(* Logix 5000 project; controller ARS14002_PLC vendor 1 type 14 code 218 rev 30.11; software revision 30.01; part 8 of 13 *)
(* tags used below, declared in another part *)
   ARS_DERIME_AUTO : BOOL;
   ARS_Manual_Backfill : BOOL;   // **future use
   ARS_RETURN_AUTO : BOOL;
   ARS_STANDBY : BOOL;
   CP_Hi_Press_Shutoff : BOOL;
   CP_PumpUp : BOOL;
   CP_PumpUp_DN_ONS_OB : BOOL;
   CP_PumpUp_PressurePermissive : BOOL;
   CP_PumpUp_Standby_Press_SP_H : DINT;
   CP_PumpUp_Standby_Press_SP_L : DINT;
   CP_Run : BOOL;
   CP_Run_Atomize : BOOL;
   CP_Run_Standby : BOOL;
   CP_Select_Auto : BOOL;
   CP_Speed_SP_Atomize : REAL;
   CP_Speed_SP_Standby : DINT;
   CP_Start_Vent_TMR_PRE : DINT;
   FVR_800C_Auto : BOOL;
   FVR_800C_EN : BOOL;
   FVR_800C_FREQ_OUT : REAL;
   FVR_800C_PRIMARY : BOOL;
   FVR_800C_RUNNING : BOOL;
   FVR_800C_ST : BOOL;
   FVR_800D_Auto : BOOL;
   FVR_800D_EN : BOOL;
   FVR_800D_FREQ_OUT : REAL;
   FVR_800D_PRIMARY : BOOL;
   FVR_800D_RUNNING : BOOL;
   FVR_800D_ST : BOOL;
   HP_Shutoff_PerPump : REAL;
   HP_Shutoff_SPH : DINT;
   HP_Shutoff_SPL : DINT;
   IGNORE_TE_802S : BOOL;   // Don't look at TE_802
   MODE_ATOMIZE : BOOL;
   P_800_COOLDOWN_ALT_TIME : REAL;
   P_800_COOLDOWN_ALT_TIME_MS : DINT;
   P_800A_Cavit : BOOL;
   P_800A_CAVIT_CHK_TMR : TIMER;
   P_800A_CAVIT_CTR : COUNTER;
   P_800A_CAVIT_CTR_MONTH : COUNTER;
   P_800A_Cavit_Shutdown : BOOL;
   P_800A_CAVIT_TEMP_SP : DINT;
   P_800A_CAVIT_VENT_START_DLA_TMR : TIMER;
   P_800A_Cavit_Vent_TMR : TIMER;
   P_800A_COOLDOWN_ALT_TON : TIMER;
   P_800A_Hi_Press_Shutoff : BOOL;
   P_800A_Init_OK : BOOL;
   P_800A_Pre_Vent_Done : BOOL;
   P_800A_Pre_Vent_Pending : BOOL;
   P_800A_Prestart : BOOL;
   P_800A_Ready : BOOL;
   P_800A_Select_Auto_Online : BOOL;
   P_800A_Start_DLA_TMR : TIMER;
   P_800A_Start_TMR : TIMER;
   P_800A_Start_Vent_TMR : TIMER;
   P_800A_Stop_Vent_Delay : BOOL;
   P_800A_Stop_Vent_TMR : TIMER;
   P_800B_Cavit : BOOL;
   P_800B_CAVIT_CHK_TMR : TIMER;
   P_800B_CAVIT_CTR : COUNTER;
   P_800B_CAVIT_CTR_MONTH : COUNTER;
   P_800B_Cavit_Shutdown : BOOL;
   P_800B_CAVIT_TEMP_SP : DINT;
   P_800B_CAVIT_VENT_START_DLA_TMR : TIMER;
   P_800B_Cavit_Vent_TMR : TIMER;
   P_800B_COOLDOWN_ALT_TON : TIMER;
   P_800B_Hi_Press_Shutoff : BOOL;
   P_800B_Init_OK : BOOL;
   P_800B_Pre_Vent_Done : BOOL;
   P_800B_Pre_Vent_Pending : BOOL;
   P_800B_Prestart : BOOL;
   P_800B_Ready : BOOL;
   P_800B_Select_Auto_Online : BOOL;
   P_800B_Start_DLA_TMR : TIMER;
   P_800B_Start_TMR : TIMER;
   P_800B_Start_Vent_TMR : TIMER;
   P_800B_Stop_Vent_Delay : BOOL;
   P_800B_Stop_Vent_TMR : TIMER;
   P_800C : CM_DO_FVR;
   P_800C_Cavit : BOOL;
   P_800C_CAVIT_CHK_TMR : TIMER;
   P_800C_CAVIT_CTR : COUNTER;
   P_800C_CAVIT_CTR_MONTH : COUNTER;
   P_800C_Cavit_Shutdown : BOOL;
   P_800C_CAVIT_TEMP_SP : DINT;
   P_800C_CAVIT_VENT_START_DLA_TMR : TIMER;
   P_800C_Cavit_Vent_TMR : TIMER;
   P_800C_COOLDOWN_ALT_TON : TIMER;
   P_800C_Fault : BOOL;
   P_800C_Hi_Press_Shutoff : BOOL;
   P_800C_Init_OK : BOOL;
   P_800C_Pre_Vent_Done : BOOL;
   P_800C_Pre_Vent_Pending : BOOL;
   P_800C_Prestart : BOOL;
   P_800C_Ready : BOOL;
   P_800C_Start_DLA_TMR : TIMER;
   P_800C_Start_TMR : TIMER;
   P_800C_Start_Vent_TMR : TIMER;
   P_800C_Stop_Vent_Delay : BOOL;
   P_800C_Stop_Vent_TMR : TIMER;
   P_800D : CM_DO_FVR;
   P_800D_Cavit : BOOL;
   P_800D_CAVIT_CHK_TMR : TIMER;
   P_800D_CAVIT_CTR : COUNTER;
   P_800D_CAVIT_CTR_MONTH : COUNTER;
   P_800D_Cavit_Shutdown : BOOL;
   P_800D_CAVIT_TEMP_SP : DINT;
   P_800D_CAVIT_VENT_START_DLA_TMR : TIMER;
   P_800D_Cavit_Vent_TMR : TIMER;
   P_800D_COOLDOWN_ALT_TON : TIMER;
   P_800D_Fault : BOOL;
   P_800D_Hi_Press_Shutoff : BOOL;
   P_800D_Init_OK : BOOL;
   P_800D_Pre_Vent_Done : BOOL;
   P_800D_Pre_Vent_Pending : BOOL;
   P_800D_Prestart : BOOL;
   P_800D_Ready : BOOL;
   P_800D_Start_DLA_TMR : TIMER;
   P_800D_Start_Temp_SP : DINT;
   P_800D_Start_TMR : TIMER;
   P_800D_Start_Vent_TMR : TIMER;
   P_800D_Stop_Vent_Delay : BOOL;
   P_800D_Stop_Vent_TMR : TIMER;
   PDT_751 : CM_AI_SCL_ALT;
   PIDE_800 : PID_ENHANCED;
   PIDE_800_CVOper_HZ : REAL;
   PIDE_800_CVProg_HZ : REAL;
   PIDE_800_OPER_ONS : BOOL;
   PT_802A : CM_AI_SCL;
   PT_802B : CM_AI_SCL;
   PT_802C : CM_AI_SCL;
   PT_802D : CM_AI_SCL;
   PT_806 : CM_AI_SCL;
   PT_902 : CM_AI_SCL;
   PUMP_CALC_FLOW : REAL;
   PUMP_CAVIT_PRESSURE_MARGIN : REAL;   // HOW MUCH LOWER PUMP PT CAN BE THAN PT-902
   PUMP_CAVIT_PRESSURE_SP : REAL;
   PWHMI_StartAtomizing : TIMER;
   START_ATOMIZE_DURING_PUMPUP : BOOL;
   SV_802AX : CM_DO_GENERIC;
   SV_802BX : CM_DO_GENERIC;
   SV_802CX : CM_DO_GENERIC;
   SV_802DX : CM_DO_GENERIC;
   TE_802_INIT_TEMP : REAL;
   TE_802A : CM_AI_SCL;
   TE_802B : CM_AI_SCL;
   TE_802C : CM_AI_SCL;
   TE_802D : CM_AI_SCL;
   TE_803D : CM_AI_SCL;
   TE_804_INIT_TEMP : REAL;
   TE_804A : CM_AI_SCL;
   TE_804B : CM_AI_SCL;
   TE_804C : CM_AI_SCL;
   TE_804D : CM_AI_SCL;
   TEST_COOLDOWN_ALT : BOOL;
   VFD_800A_Auto : BOOL;
   VFD_800A_EN : BOOL;
   VFD_800A_ST : BOOL;
   VFD_800B_Auto : BOOL;
   VFD_800B_EN : BOOL;
   VFD_800B_ST : BOOL;
   XV_806 : CM_DO_VLV;
   XV_806_SPH_802_CLOSED : REAL;
   XV_806_SPH_802_OPEN : REAL;
   XV_806_SPL_802_CLOSED : REAL;
   XV_806_SPL_802_OPEN : REAL;
(* MainProgram, continued *)

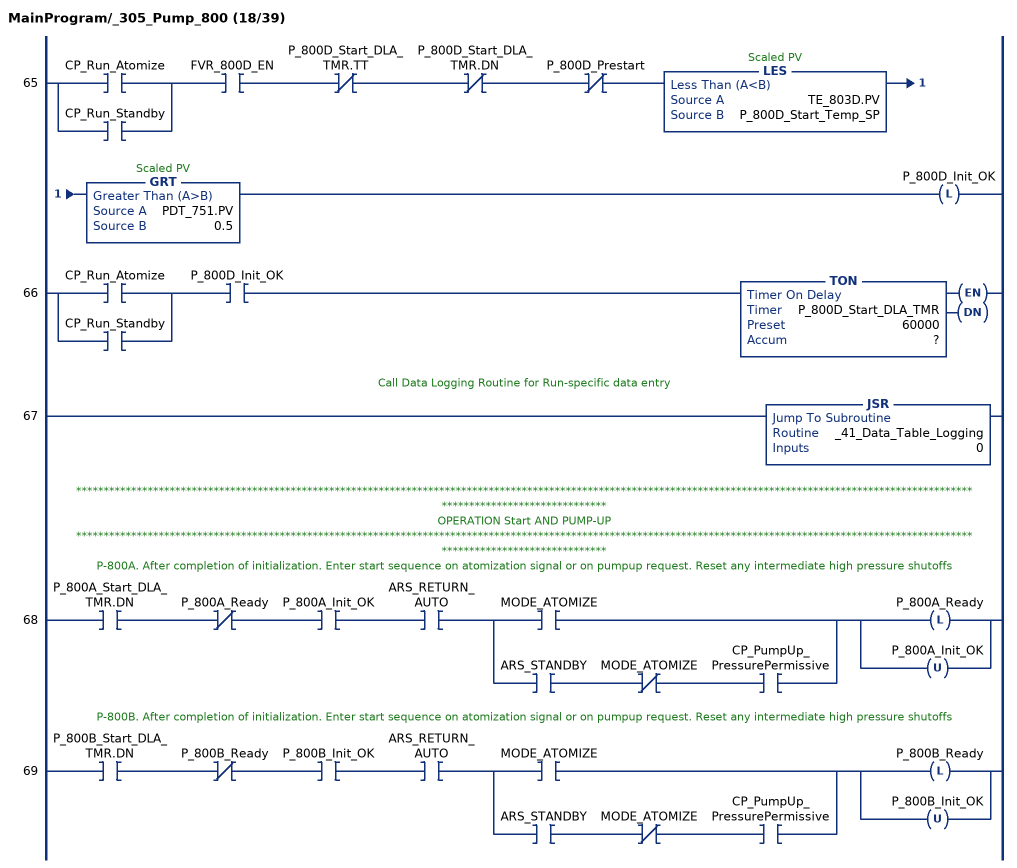
   [picture p154: MainProgram/_305_Pump_800 rungs 65-69]
   65: [XIC(CP_Run_Atomize) ,XIC(CP_Run_Standby) ]XIC(FVR_800D_EN)XIO(P_800D_Start_DLA_TMR.TT)XIO(P_800D_Start_DLA_TMR.DN)XIO(P_800D_Prestart)LES(TE_803D.PV,P_800D_Start_Temp_SP)GRT(PDT_751.PV,0.5)OTL(P_800D_Init_OK);
   66: [XIC(CP_Run_Atomize) ,XIC(CP_Run_Standby) ]XIC(P_800D_Init_OK)TON(P_800D_Start_DLA_TMR,?,?);
   // Call Data Logging Routine for Run-specific data entry
   67: JSR(_41_Data_Table_Logging,0);
   // *************************************************************************************************************************************************************************************************
   // OPERATION Start AND PUMP-UP
   // *************************************************************************************************************************************************************************************************
   // P-800A. After completion of initialization. Enter start sequence on atomization signal or on pumpup request. Reset any intermediate high pressure shutoffs
   68: XIC(P_800A_Start_DLA_TMR.DN)XIO(P_800A_Ready)XIC(P_800A_Init_OK)XIC(ARS_RETURN_AUTO)[XIC(MODE_ATOMIZE) ,XIC(ARS_STANDBY) XIO(MODE_ATOMIZE) XIC(CP_PumpUp_PressurePermissive) ][OTL(P_800A_Ready) ,OTU(P_800A_Init_OK) ];
   // P-800B. After completion of initialization. Enter start sequence on atomization signal or on pumpup request. Reset any intermediate high pressure shutoffs
   69: XIC(P_800B_Start_DLA_TMR.DN)XIO(P_800B_Ready)XIC(P_800B_Init_OK)XIC(ARS_RETURN_AUTO)[XIC(MODE_ATOMIZE) ,XIC(ARS_STANDBY) XIO(MODE_ATOMIZE) XIC(CP_PumpUp_PressurePermissive) ][OTL(P_800B_Ready) ,OTU(P_800B_Init_OK) ];
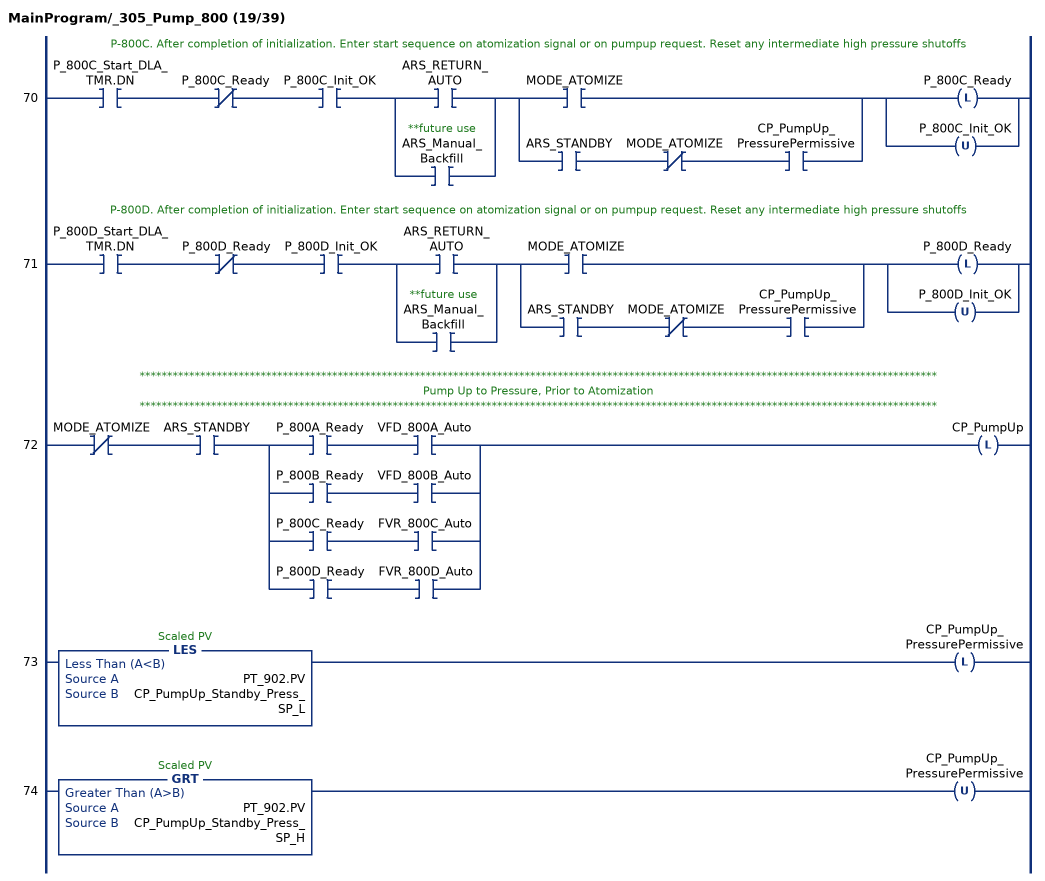
   // P-800C. After completion of initialization. Enter start sequence on atomization signal or on pumpup request. Reset any intermediate high pressure shutoffs
   70: XIC(P_800C_Start_DLA_TMR.DN)XIO(P_800C_Ready)XIC(P_800C_Init_OK)[XIC(ARS_RETURN_AUTO) ,XIC(ARS_Manual_Backfill) ][XIC(MODE_ATOMIZE) ,XIC(ARS_STANDBY) XIO(MODE_ATOMIZE) XIC(CP_PumpUp_PressurePermissive) ][OTL(P_800C_Ready) ,OTU(P_800C_Init_OK) ];
   // P-800D. After completion of initialization. Enter start sequence on atomization signal or on pumpup request. Reset any intermediate high pressure shutoffs
   71: XIC(P_800D_Start_DLA_TMR.DN)XIO(P_800D_Ready)XIC(P_800D_Init_OK)[XIC(ARS_RETURN_AUTO) ,XIC(ARS_Manual_Backfill) ][XIC(MODE_ATOMIZE) ,XIC(ARS_STANDBY) XIO(MODE_ATOMIZE) XIC(CP_PumpUp_PressurePermissive) ][OTL(P_800D_Ready) ,OTU(P_800D_Init_OK) ];
   // *************************************************************************************************************************************************
   // Pump Up to Pressure, Prior to Atomization
   // *************************************************************************************************************************************************
   72: XIO(MODE_ATOMIZE)XIC(ARS_STANDBY)[XIC(P_800A_Ready) XIC(VFD_800A_Auto) ,XIC(P_800B_Ready) XIC(VFD_800B_Auto) ,XIC(P_800C_Ready) XIC(FVR_800C_Auto) ,XIC(P_800D_Ready) XIC(FVR_800D_Auto) ]OTL(CP_PumpUp);
   73: LES(PT_902.PV,CP_PumpUp_Standby_Press_SP_L)OTL(CP_PumpUp_PressurePermissive);
   74: GRT(PT_902.PV,CP_PumpUp_Standby_Press_SP_H)OTU(CP_PumpUp_PressurePermissive);
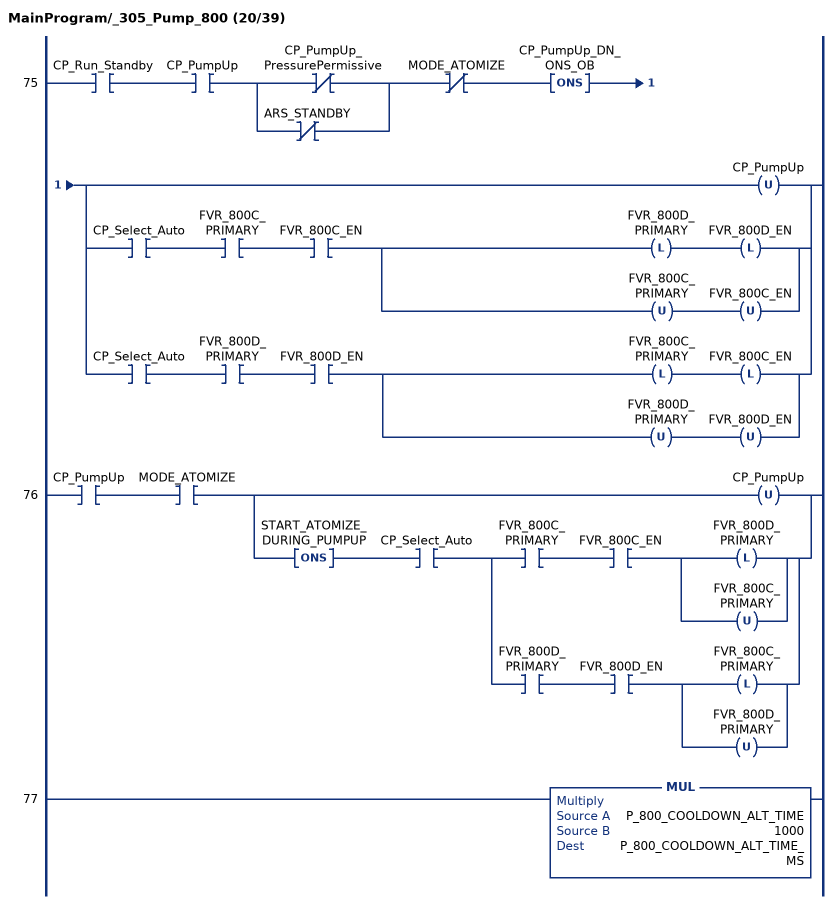
   75: XIC(CP_Run_Standby)XIC(CP_PumpUp)[XIO(CP_PumpUp_PressurePermissive) ,XIO(ARS_STANDBY) ]XIO(MODE_ATOMIZE)ONS(CP_PumpUp_DN_ONS_OB)[[OTU(CP_PumpUp) ,XIC(CP_Select_Auto) XIC(FVR_800C_PRIMARY) XIC(FVR_800C_EN) [OTL(FVR_800D_PRIMARY) OTL(FVR_800D_EN) ,OTU(FVR_800C_PRIMARY) OTU(FVR_800C_EN) ] ] ,XIC(CP_Select_Auto) XIC(FVR_800D_PRIMARY) XIC(FVR_800D_EN) [OTL(FVR_800C_PRIMARY) OTL(FVR_800C_EN) ,OTU(FVR_800D_PRIMARY) OTU(FVR_800D_EN) ] ];
   76: XIC(CP_PumpUp)XIC(MODE_ATOMIZE)[OTU(CP_PumpUp) ,ONS(START_ATOMIZE_DURING_PUMPUP) XIC(CP_Select_Auto) [XIC(FVR_800C_PRIMARY) XIC(FVR_800C_EN) [OTL(FVR_800D_PRIMARY) ,OTU(FVR_800C_PRIMARY) ] ,XIC(FVR_800D_PRIMARY) XIC(FVR_800D_EN) [OTL(FVR_800C_PRIMARY) ,OTU(FVR_800D_PRIMARY) ] ] ];
   77: MUL(P_800_COOLDOWN_ALT_TIME,1000,P_800_COOLDOWN_ALT_TIME_MS);
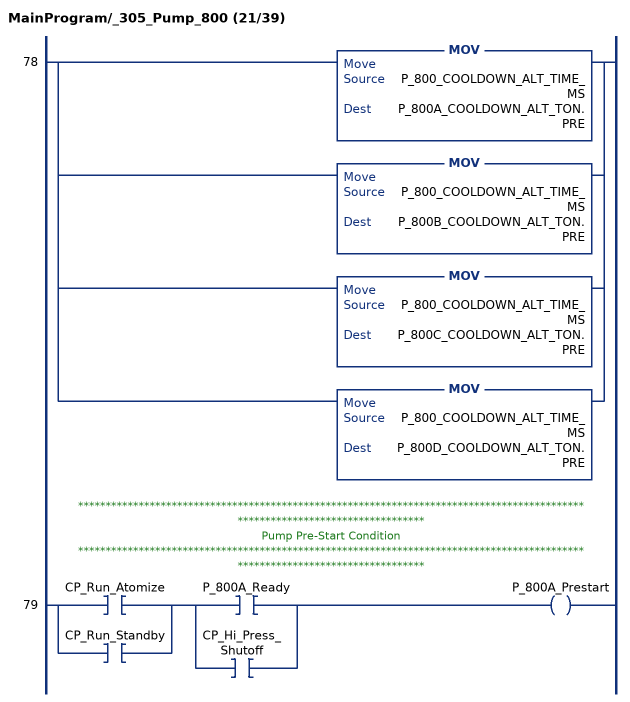
   78: [MOV(P_800_COOLDOWN_ALT_TIME_MS,P_800A_COOLDOWN_ALT_TON.PRE) ,MOV(P_800_COOLDOWN_ALT_TIME_MS,P_800B_COOLDOWN_ALT_TON.PRE) ,MOV(P_800_COOLDOWN_ALT_TIME_MS,P_800C_COOLDOWN_ALT_TON.PRE) ,MOV(P_800_COOLDOWN_ALT_TIME_MS,P_800D_COOLDOWN_ALT_TON.PRE) ];
   // ******************************************************************************************************************************
   // Pump Pre-Start Condition
   // ******************************************************************************************************************************
   79: [XIC(CP_Run_Atomize) ,XIC(CP_Run_Standby) ][XIC(P_800A_Ready) ,XIC(CP_Hi_Press_Shutoff) ]OTE(P_800A_Prestart);
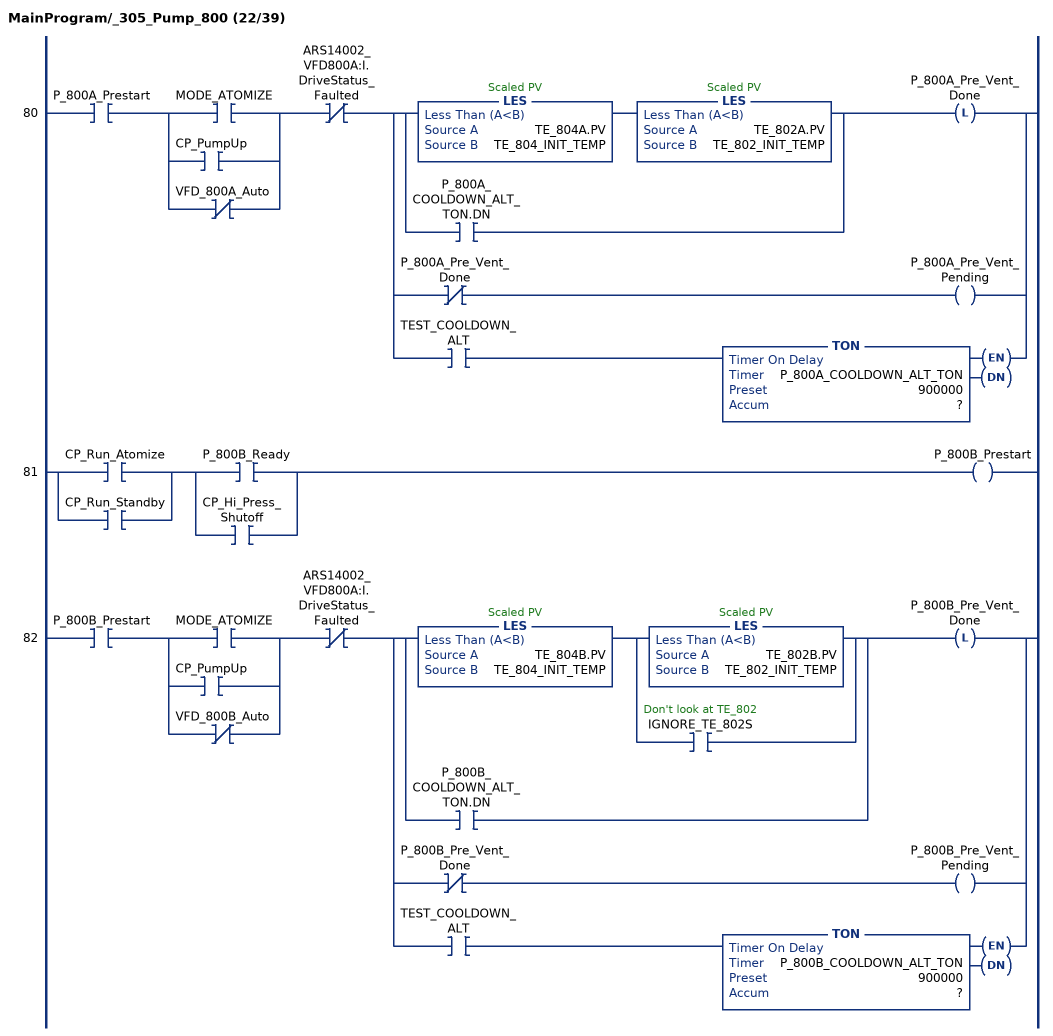
   80: XIC(P_800A_Prestart)[XIC(MODE_ATOMIZE) ,XIC(CP_PumpUp) ,XIO(VFD_800A_Auto) ]XIO(ARS14002_VFD800A:I.DriveStatus_Faulted)[[LES(TE_804A.PV,TE_804_INIT_TEMP) LES(TE_802A.PV,TE_802_INIT_TEMP) ,XIC(P_800A_COOLDOWN_ALT_TON.DN) ] OTL(P_800A_Pre_Vent_Done) ,XIO(P_800A_Pre_Vent_Done) OTE(P_800A_Pre_Vent_Pending) ,XIC(TEST_COOLDOWN_ALT) TON(P_800A_COOLDOWN_ALT_TON,?,?) ];
   81: [XIC(CP_Run_Atomize) ,XIC(CP_Run_Standby) ][XIC(P_800B_Ready) ,XIC(CP_Hi_Press_Shutoff) ]OTE(P_800B_Prestart);
   82: XIC(P_800B_Prestart)[XIC(MODE_ATOMIZE) ,XIC(CP_PumpUp) ,XIO(VFD_800B_Auto) ]XIO(ARS14002_VFD800A:I.DriveStatus_Faulted)[[LES(TE_804B.PV,TE_804_INIT_TEMP) [LES(TE_802B.PV,TE_802_INIT_TEMP) ,XIC(IGNORE_TE_802S) ] ,XIC(P_800B_COOLDOWN_ALT_TON.DN) ] OTL(P_800B_Pre_Vent_Done) ,XIO(P_800B_Pre_Vent_Done) OTE(P_800B_Pre_Vent_Pending) ,XIC(TEST_COOLDOWN_ALT) TON(P_800B_COOLDOWN_ALT_TON,?,?) ];
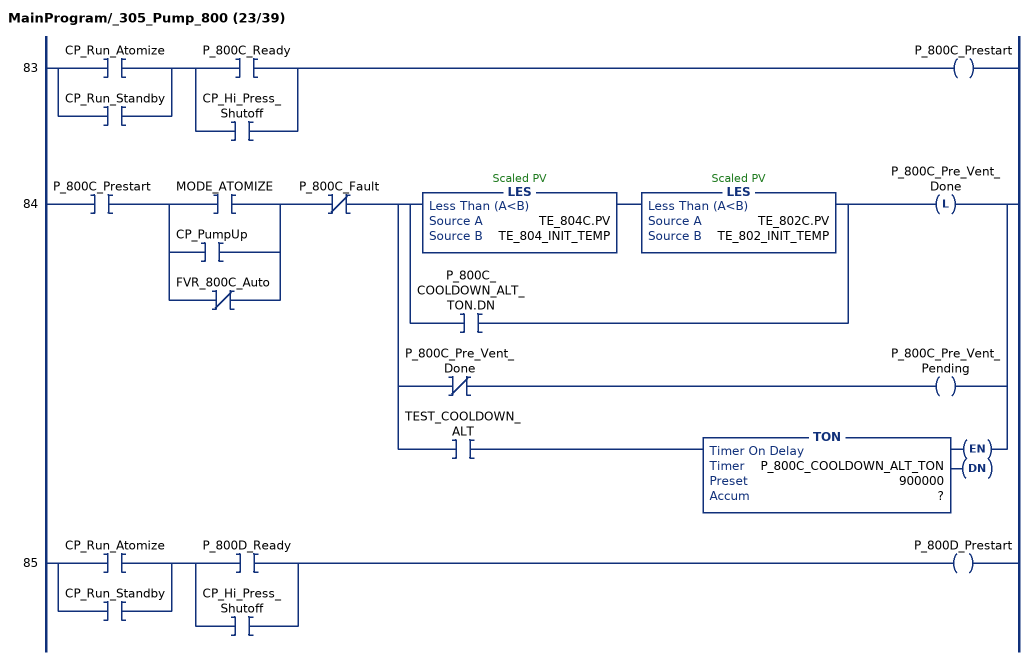
   83: [XIC(CP_Run_Atomize) ,XIC(CP_Run_Standby) ][XIC(P_800C_Ready) ,XIC(CP_Hi_Press_Shutoff) ]OTE(P_800C_Prestart);
   84: XIC(P_800C_Prestart)[XIC(MODE_ATOMIZE) ,XIC(CP_PumpUp) ,XIO(FVR_800C_Auto) ]XIO(P_800C_Fault)[[LES(TE_804C.PV,TE_804_INIT_TEMP) LES(TE_802C.PV,TE_802_INIT_TEMP) ,XIC(P_800C_COOLDOWN_ALT_TON.DN) ] OTL(P_800C_Pre_Vent_Done) ,XIO(P_800C_Pre_Vent_Done) OTE(P_800C_Pre_Vent_Pending) ,XIC(TEST_COOLDOWN_ALT) TON(P_800C_COOLDOWN_ALT_TON,?,?) ];
   85: [XIC(CP_Run_Atomize) ,XIC(CP_Run_Standby) ][XIC(P_800D_Ready) ,XIC(CP_Hi_Press_Shutoff) ]OTE(P_800D_Prestart);
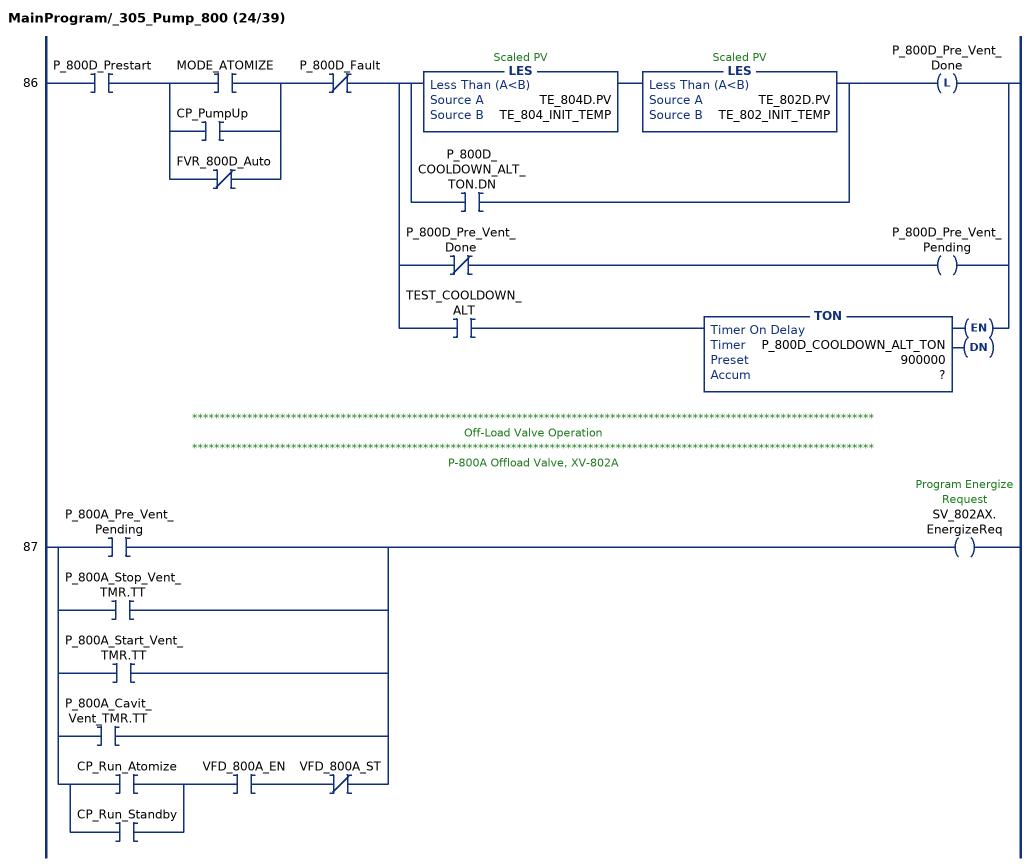
   86: XIC(P_800D_Prestart)[XIC(MODE_ATOMIZE) ,XIC(CP_PumpUp) ,XIO(FVR_800D_Auto) ]XIO(P_800D_Fault)[[LES(TE_804D.PV,TE_804_INIT_TEMP) LES(TE_802D.PV,TE_802_INIT_TEMP) ,XIC(P_800D_COOLDOWN_ALT_TON.DN) ] OTL(P_800D_Pre_Vent_Done) ,XIO(P_800D_Pre_Vent_Done) OTE(P_800D_Pre_Vent_Pending) ,XIC(TEST_COOLDOWN_ALT) TON(P_800D_COOLDOWN_ALT_TON,?,?) ];
   // ****************************************************************************************************************************
   // Off-Load Valve Operation
   // ****************************************************************************************************************************
   // P-800A Offload Valve, XV-802A
   87: [XIC(P_800A_Pre_Vent_Pending) ,XIC(P_800A_Stop_Vent_TMR.TT) ,XIC(P_800A_Start_Vent_TMR.TT) ,XIC(P_800A_Cavit_Vent_TMR.TT) ,[XIC(CP_Run_Atomize) ,XIC(CP_Run_Standby) ] XIC(VFD_800A_EN) XIO(VFD_800A_ST) ]OTE(SV_802AX.EnergizeReq);
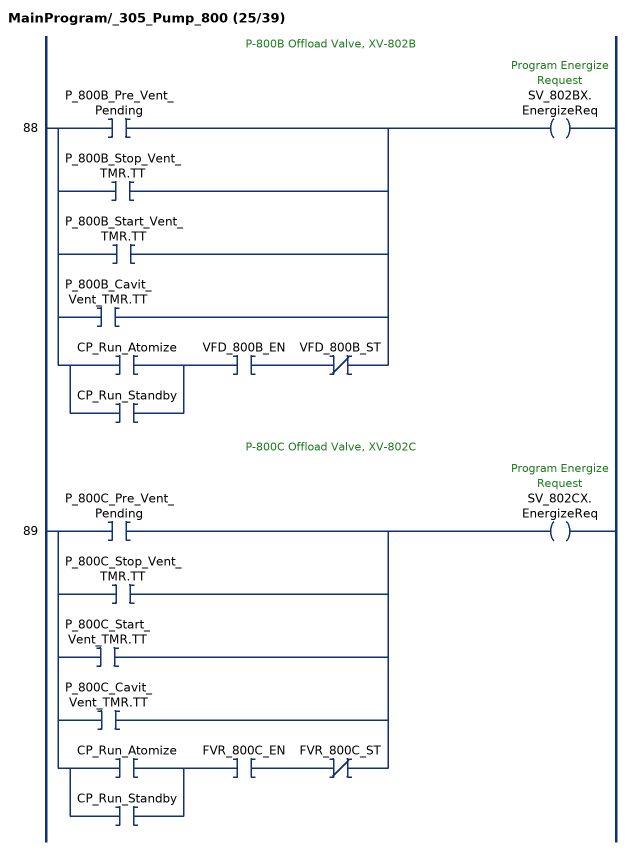
   // P-800B Offload Valve, XV-802B
   88: [XIC(P_800B_Pre_Vent_Pending) ,XIC(P_800B_Stop_Vent_TMR.TT) ,XIC(P_800B_Start_Vent_TMR.TT) ,XIC(P_800B_Cavit_Vent_TMR.TT) ,[XIC(CP_Run_Atomize) ,XIC(CP_Run_Standby) ] XIC(VFD_800B_EN) XIO(VFD_800B_ST) ]OTE(SV_802BX.EnergizeReq);
   // P-800C Offload Valve, XV-802C
   89: [XIC(P_800C_Pre_Vent_Pending) ,XIC(P_800C_Stop_Vent_TMR.TT) ,XIC(P_800C_Start_Vent_TMR.TT) ,XIC(P_800C_Cavit_Vent_TMR.TT) ,[XIC(CP_Run_Atomize) ,XIC(CP_Run_Standby) ] XIC(FVR_800C_EN) XIO(FVR_800C_ST) ]OTE(SV_802CX.EnergizeReq);
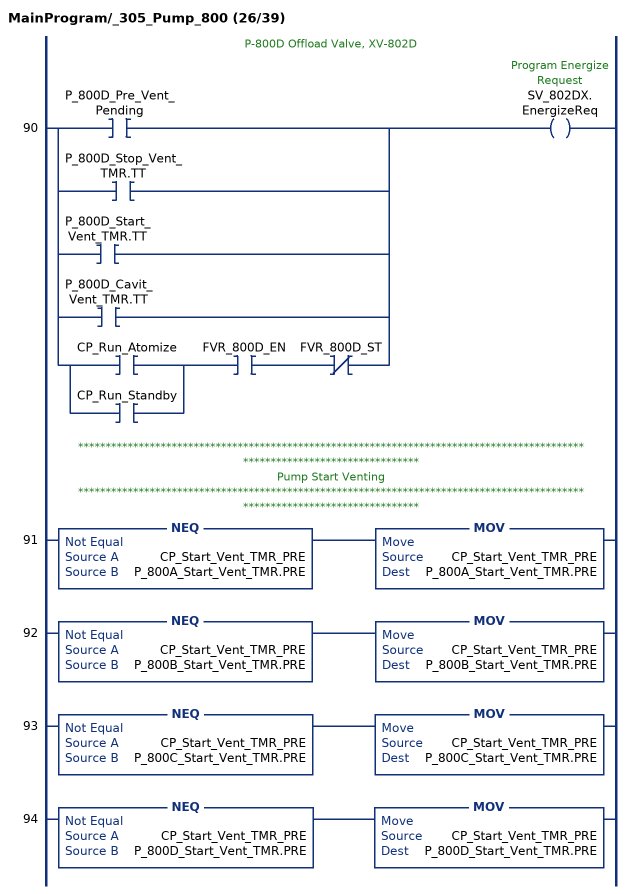
   // P-800D Offload Valve, XV-802D
   90: [XIC(P_800D_Pre_Vent_Pending) ,XIC(P_800D_Stop_Vent_TMR.TT) ,XIC(P_800D_Start_Vent_TMR.TT) ,XIC(P_800D_Cavit_Vent_TMR.TT) ,[XIC(CP_Run_Atomize) ,XIC(CP_Run_Standby) ] XIC(FVR_800D_EN) XIO(FVR_800D_ST) ]OTE(SV_802DX.EnergizeReq);
   // ****************************************************************************************************************************
   // Pump Start Venting
   // ****************************************************************************************************************************
   91: NEQ(CP_Start_Vent_TMR_PRE,P_800A_Start_Vent_TMR.PRE)MOV(CP_Start_Vent_TMR_PRE,P_800A_Start_Vent_TMR.PRE);
   92: NEQ(CP_Start_Vent_TMR_PRE,P_800B_Start_Vent_TMR.PRE)MOV(CP_Start_Vent_TMR_PRE,P_800B_Start_Vent_TMR.PRE);
   93: NEQ(CP_Start_Vent_TMR_PRE,P_800C_Start_Vent_TMR.PRE)MOV(CP_Start_Vent_TMR_PRE,P_800C_Start_Vent_TMR.PRE);
   94: NEQ(CP_Start_Vent_TMR_PRE,P_800D_Start_Vent_TMR.PRE)MOV(CP_Start_Vent_TMR_PRE,P_800D_Start_Vent_TMR.PRE);
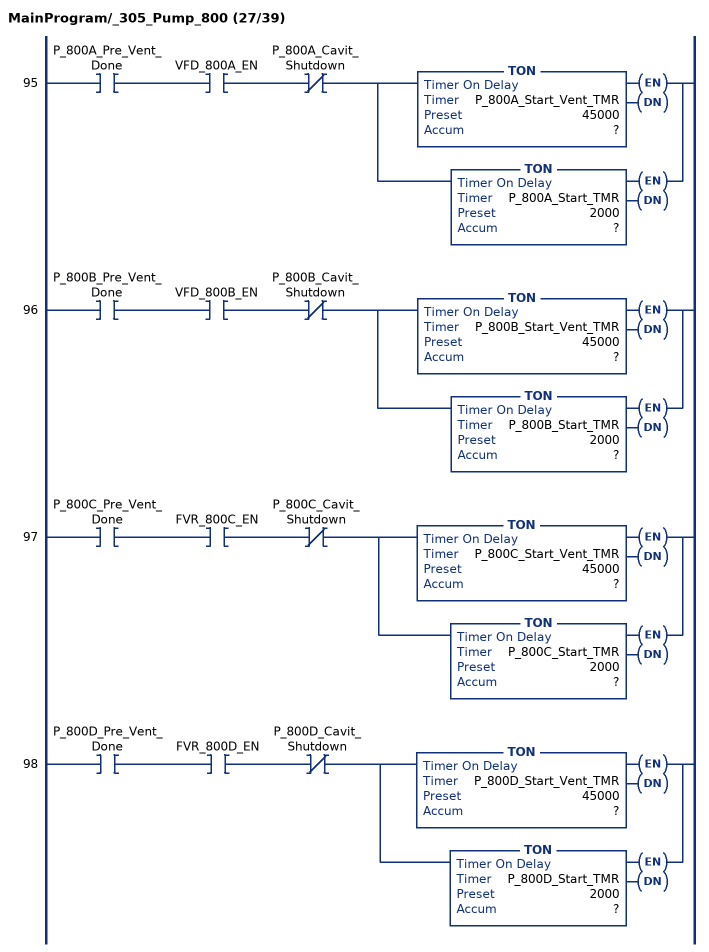
   95: XIC(P_800A_Pre_Vent_Done)XIC(VFD_800A_EN)XIO(P_800A_Cavit_Shutdown)[TON(P_800A_Start_Vent_TMR,?,?) ,TON(P_800A_Start_TMR,?,?) ];
   96: XIC(P_800B_Pre_Vent_Done)XIC(VFD_800B_EN)XIO(P_800B_Cavit_Shutdown)[TON(P_800B_Start_Vent_TMR,?,?) ,TON(P_800B_Start_TMR,?,?) ];
   97: XIC(P_800C_Pre_Vent_Done)XIC(FVR_800C_EN)XIO(P_800C_Cavit_Shutdown)[TON(P_800C_Start_Vent_TMR,?,?) ,TON(P_800C_Start_TMR,?,?) ];
   98: XIC(P_800D_Pre_Vent_Done)XIC(FVR_800D_EN)XIO(P_800D_Cavit_Shutdown)[TON(P_800D_Start_Vent_TMR,?,?) ,TON(P_800D_Start_TMR,?,?) ];
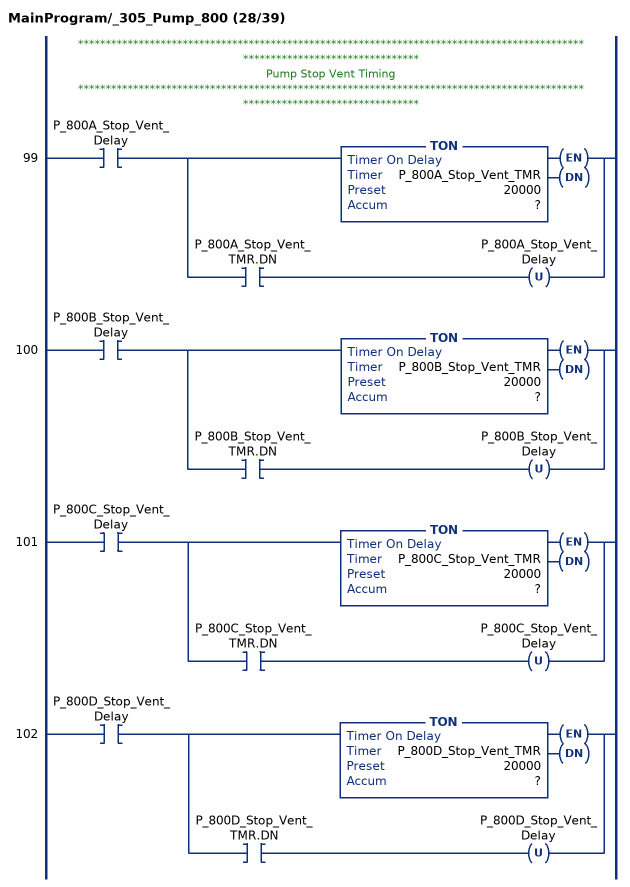
   // ****************************************************************************************************************************
   // Pump Stop Vent Timing
   // ****************************************************************************************************************************
   99: XIC(P_800A_Stop_Vent_Delay)[TON(P_800A_Stop_Vent_TMR,?,?) ,XIC(P_800A_Stop_Vent_TMR.DN) OTU(P_800A_Stop_Vent_Delay) ];
   100: XIC(P_800B_Stop_Vent_Delay)[TON(P_800B_Stop_Vent_TMR,?,?) ,XIC(P_800B_Stop_Vent_TMR.DN) OTU(P_800B_Stop_Vent_Delay) ];
   101: XIC(P_800C_Stop_Vent_Delay)[TON(P_800C_Stop_Vent_TMR,?,?) ,XIC(P_800C_Stop_Vent_TMR.DN) OTU(P_800C_Stop_Vent_Delay) ];
   102: XIC(P_800D_Stop_Vent_Delay)[TON(P_800D_Stop_Vent_TMR,?,?) ,XIC(P_800D_Stop_Vent_TMR.DN) OTU(P_800D_Stop_Vent_Delay) ];
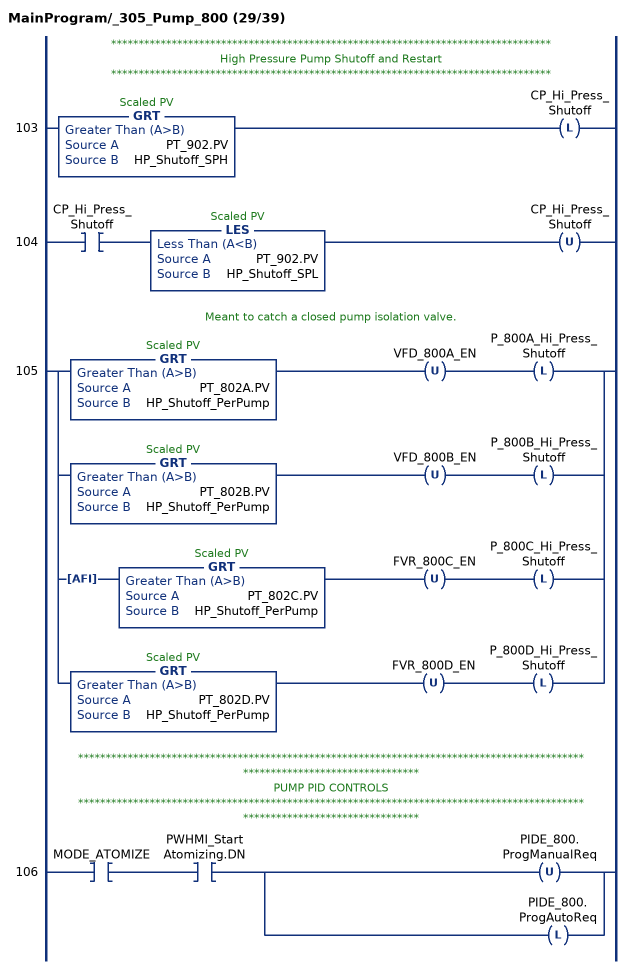
   // ********************************************************************************
   // High Pressure Pump Shutoff and Restart
   // ********************************************************************************
   103: GRT(PT_902.PV,HP_Shutoff_SPH)OTL(CP_Hi_Press_Shutoff);
   104: XIC(CP_Hi_Press_Shutoff)LES(PT_902.PV,HP_Shutoff_SPL)OTU(CP_Hi_Press_Shutoff);
   // Meant to catch a closed pump isolation valve.
   105: [GRT(PT_802A.PV,HP_Shutoff_PerPump) OTU(VFD_800A_EN) OTL(P_800A_Hi_Press_Shutoff) ,GRT(PT_802B.PV,HP_Shutoff_PerPump) OTU(VFD_800B_EN) OTL(P_800B_Hi_Press_Shutoff) ,AFI() GRT(PT_802C.PV,HP_Shutoff_PerPump) OTU(FVR_800C_EN) OTL(P_800C_Hi_Press_Shutoff) ,GRT(PT_802D.PV,HP_Shutoff_PerPump) OTU(FVR_800D_EN) OTL(P_800D_Hi_Press_Shutoff) ];
   // ****************************************************************************************************************************
   // PUMP PID CONTROLS
   // ****************************************************************************************************************************
   106: XIC(MODE_ATOMIZE)XIC(PWHMI_StartAtomizing.DN)[OTU(PIDE_800.ProgManualReq) ,OTL(PIDE_800.ProgAutoReq) ];
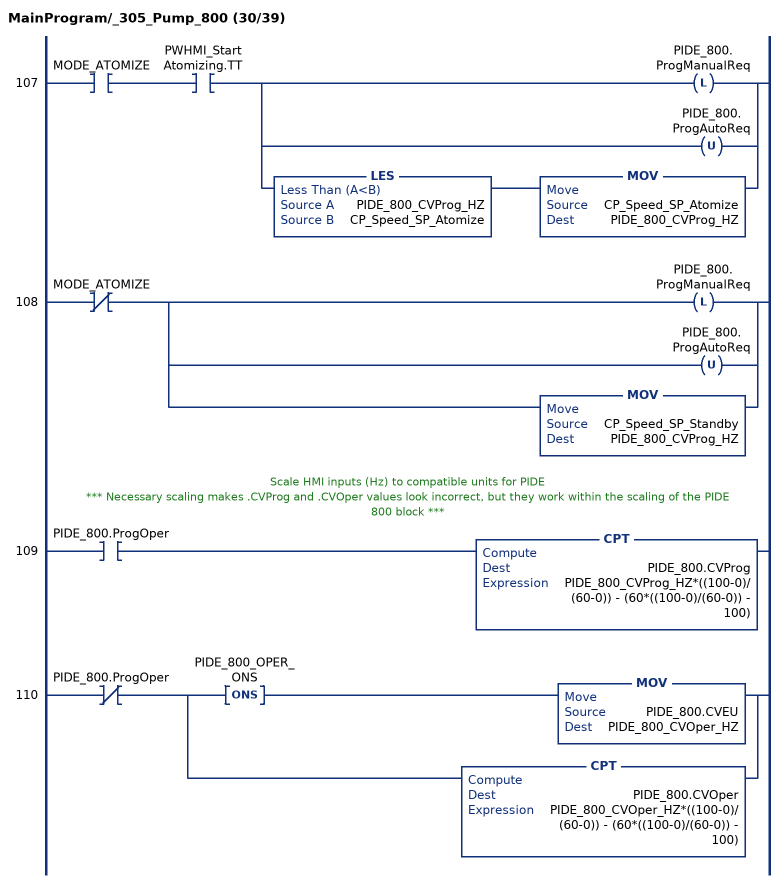
   107: XIC(MODE_ATOMIZE)XIC(PWHMI_StartAtomizing.TT)[OTL(PIDE_800.ProgManualReq) ,OTU(PIDE_800.ProgAutoReq) ,LES(PIDE_800_CVProg_HZ,CP_Speed_SP_Atomize) MOV(CP_Speed_SP_Atomize,PIDE_800_CVProg_HZ) ];
   108: XIO(MODE_ATOMIZE)[[OTL(PIDE_800.ProgManualReq) ,OTU(PIDE_800.ProgAutoReq) ] ,MOV(CP_Speed_SP_Standby,PIDE_800_CVProg_HZ) ];
   // Scale HMI inputs (Hz) to compatible units for PIDE
   // *** Necessary scaling makes .CVProg and .CVOper values look incorrect, but they work within the scaling of the PIDE 800 block ***
   109: XIC(PIDE_800.ProgOper)CPT(PIDE_800.CVProg,PIDE_800_CVProg_HZ*((100-0)/(60-0)) - (60*((100-0)/(60-0)) - 100));
   110: XIO(PIDE_800.ProgOper)[ONS(PIDE_800_OPER_ONS) MOV(PIDE_800.CVEU,PIDE_800_CVOper_HZ) ,CPT(PIDE_800.CVOper,PIDE_800_CVOper_HZ*((100-0)/(60-0)) - (60*((100-0)/(60-0)) - 100)) ];
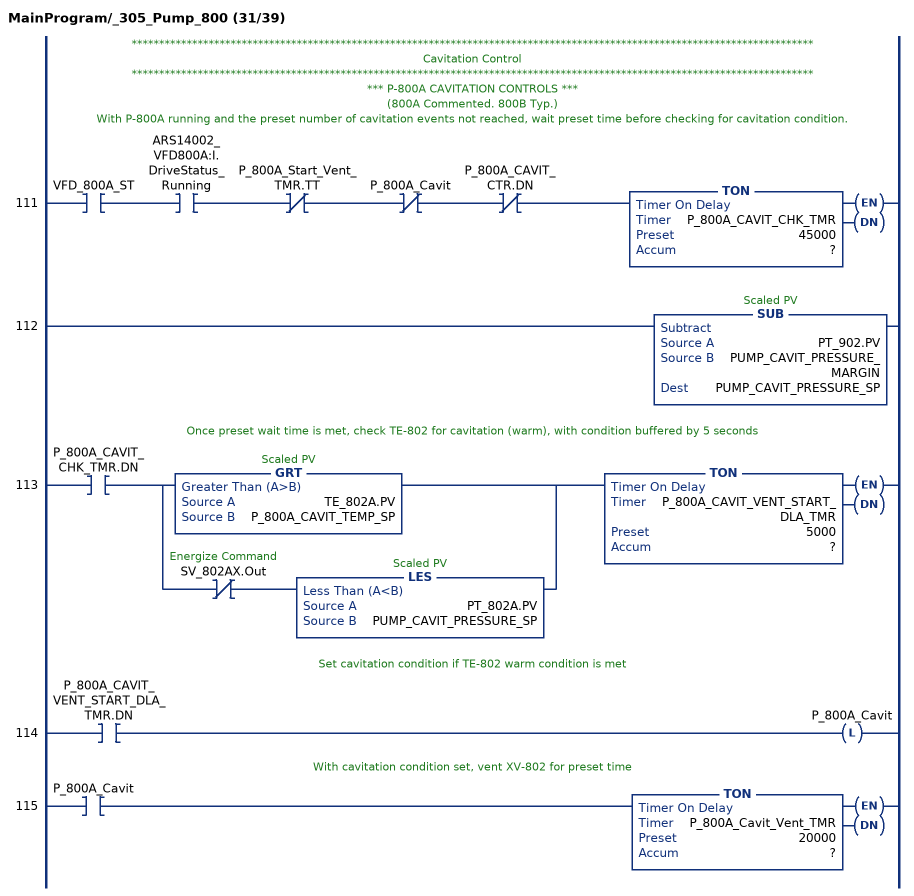
   // ****************************************************************************************************************************
   // Cavitation Control
   // ****************************************************************************************************************************
   // *** P-800A CAVITATION CONTROLS ***
   // (800A Commented. 800B Typ.)
   // With P-800A running and the preset number of cavitation events not reached, wait preset time before checking for cavitation condition.
   111: XIC(VFD_800A_ST)XIC(ARS14002_VFD800A:I.DriveStatus_Running)XIO(P_800A_Start_Vent_TMR.TT)XIO(P_800A_Cavit)XIO(P_800A_CAVIT_CTR.DN)TON(P_800A_CAVIT_CHK_TMR,?,?);
   112: SUB(PT_902.PV,PUMP_CAVIT_PRESSURE_MARGIN,PUMP_CAVIT_PRESSURE_SP);
   // Once preset wait time is met, check TE-802 for cavitation (warm), with condition buffered by 5 seconds
   113: XIC(P_800A_CAVIT_CHK_TMR.DN)[GRT(TE_802A.PV,P_800A_CAVIT_TEMP_SP) ,XIO(SV_802AX.Out) LES(PT_802A.PV,PUMP_CAVIT_PRESSURE_SP) ]TON(P_800A_CAVIT_VENT_START_DLA_TMR,?,?);
   // Set cavitation condition if TE-802 warm condition is met
   114: XIC(P_800A_CAVIT_VENT_START_DLA_TMR.DN)OTL(P_800A_Cavit);
   // With cavitation condition set, vent XV-802 for preset time
   115: XIC(P_800A_Cavit)TON(P_800A_Cavit_Vent_TMR,?,?);
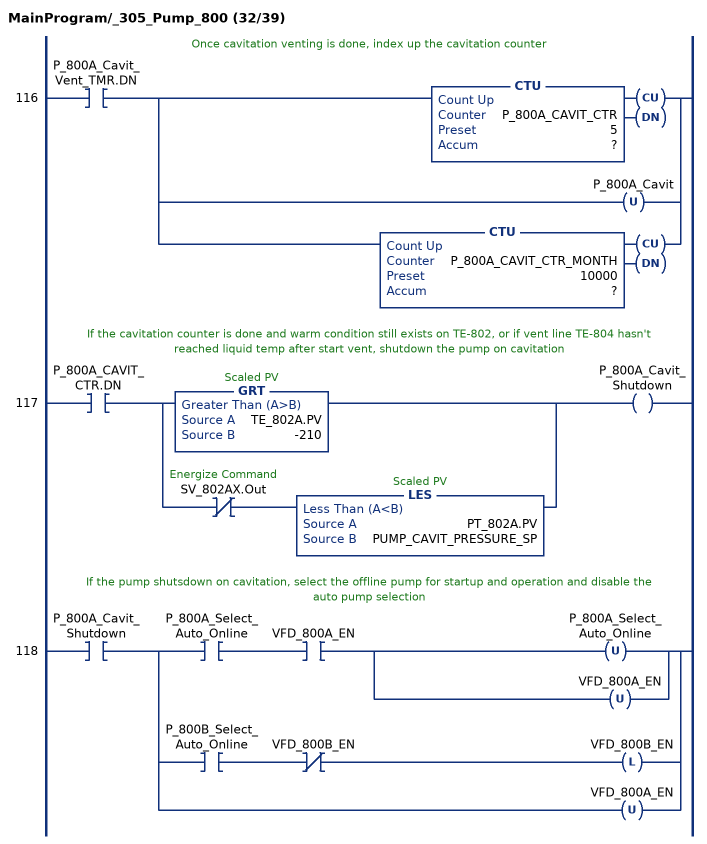
   // Once cavitation venting is done, index up the cavitation counter
   116: XIC(P_800A_Cavit_Vent_TMR.DN)[CTU(P_800A_CAVIT_CTR,?,?) ,OTU(P_800A_Cavit) ,CTU(P_800A_CAVIT_CTR_MONTH,?,?) ];
   // If the cavitation counter is done and warm condition still exists on TE-802, or if vent line TE-804 hasn't reached liquid temp after start vent, shutdown the pump on cavitation
   117: XIC(P_800A_CAVIT_CTR.DN)[GRT(TE_802A.PV,-210) ,XIO(SV_802AX.Out) LES(PT_802A.PV,PUMP_CAVIT_PRESSURE_SP) ]OTE(P_800A_Cavit_Shutdown);
   // If the pump shutsdown on cavitation, select the offline pump for startup and operation and disable the auto pump selection
   118: XIC(P_800A_Cavit_Shutdown)[XIC(P_800A_Select_Auto_Online) XIC(VFD_800A_EN) [OTU(P_800A_Select_Auto_Online) ,OTU(VFD_800A_EN) ] ,XIC(P_800B_Select_Auto_Online) XIO(VFD_800B_EN) OTL(VFD_800B_EN) ,OTU(VFD_800A_EN) ];
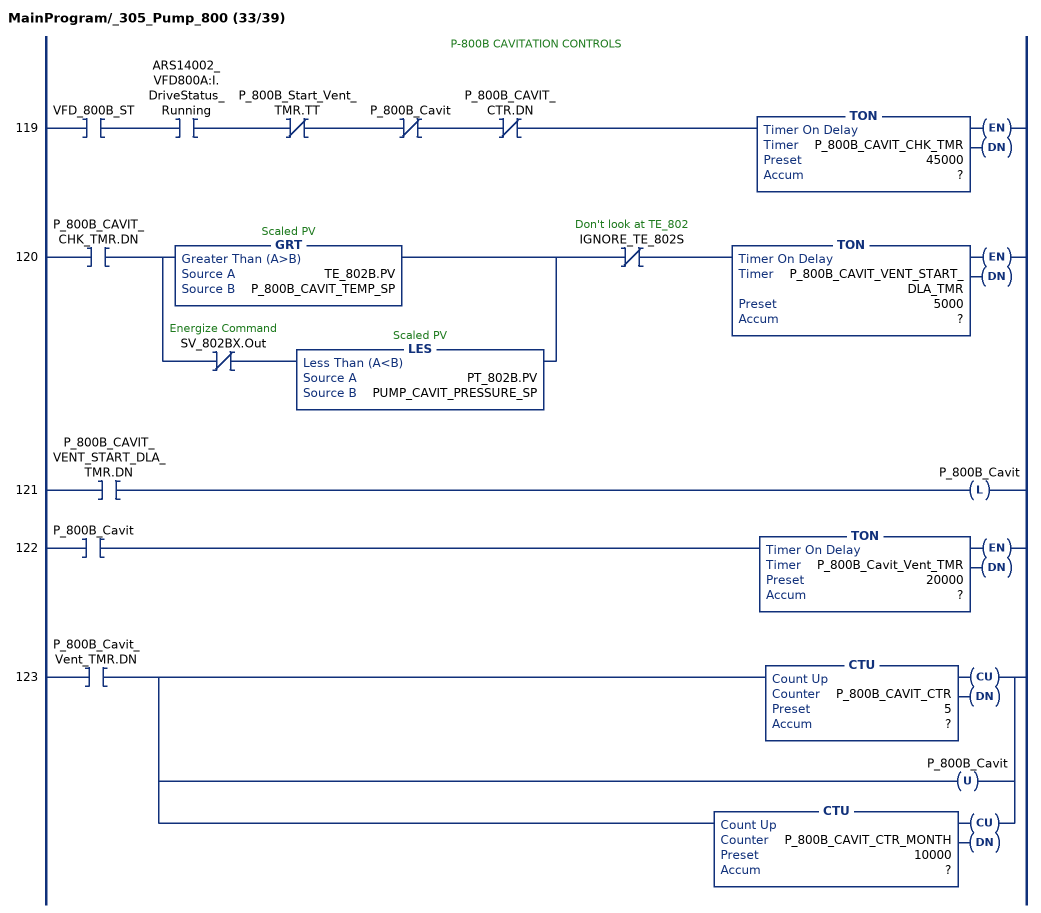
   // P-800B CAVITATION CONTROLS
   119: XIC(VFD_800B_ST)XIC(ARS14002_VFD800A:I.DriveStatus_Running)XIO(P_800B_Start_Vent_TMR.TT)XIO(P_800B_Cavit)XIO(P_800B_CAVIT_CTR.DN)TON(P_800B_CAVIT_CHK_TMR,?,?);
   120: XIC(P_800B_CAVIT_CHK_TMR.DN)[GRT(TE_802B.PV,P_800B_CAVIT_TEMP_SP) ,XIO(SV_802BX.Out) LES(PT_802B.PV,PUMP_CAVIT_PRESSURE_SP) ]XIO(IGNORE_TE_802S)TON(P_800B_CAVIT_VENT_START_DLA_TMR,?,?);
   121: XIC(P_800B_CAVIT_VENT_START_DLA_TMR.DN)OTL(P_800B_Cavit);
   122: XIC(P_800B_Cavit)TON(P_800B_Cavit_Vent_TMR,?,?);
   123: XIC(P_800B_Cavit_Vent_TMR.DN)[CTU(P_800B_CAVIT_CTR,?,?) ,OTU(P_800B_Cavit) ,CTU(P_800B_CAVIT_CTR_MONTH,?,?) ];
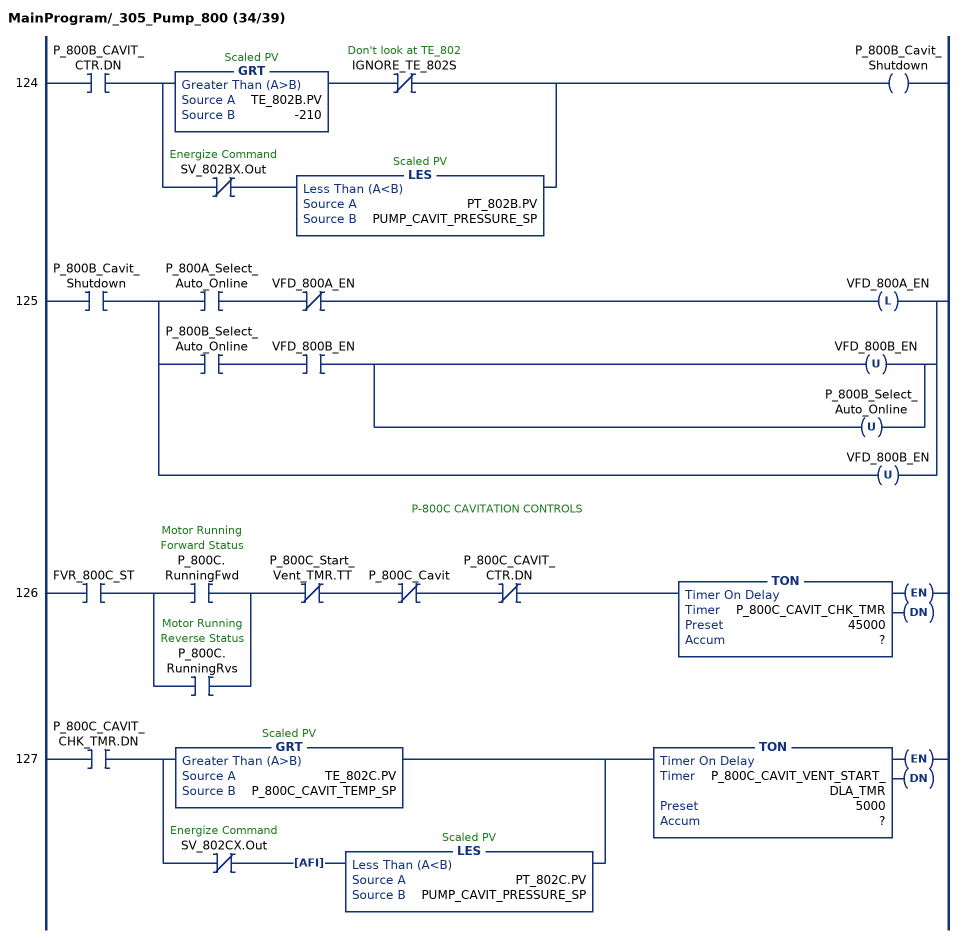
   124: XIC(P_800B_CAVIT_CTR.DN)[GRT(TE_802B.PV,-210) XIO(IGNORE_TE_802S) ,XIO(SV_802BX.Out) LES(PT_802B.PV,PUMP_CAVIT_PRESSURE_SP) ]OTE(P_800B_Cavit_Shutdown);
   125: XIC(P_800B_Cavit_Shutdown)[XIC(P_800A_Select_Auto_Online) XIO(VFD_800A_EN) OTL(VFD_800A_EN) ,XIC(P_800B_Select_Auto_Online) XIC(VFD_800B_EN) [OTU(VFD_800B_EN) ,OTU(P_800B_Select_Auto_Online) ] ,OTU(VFD_800B_EN) ];
   // P-800C CAVITATION CONTROLS
   126: XIC(FVR_800C_ST)[XIC(P_800C.RunningFwd) ,XIC(P_800C.RunningRvs) ]XIO(P_800C_Start_Vent_TMR.TT)XIO(P_800C_Cavit)XIO(P_800C_CAVIT_CTR.DN)TON(P_800C_CAVIT_CHK_TMR,?,?);
   127: XIC(P_800C_CAVIT_CHK_TMR.DN)[GRT(TE_802C.PV,P_800C_CAVIT_TEMP_SP) ,XIO(SV_802CX.Out) AFI() LES(PT_802C.PV,PUMP_CAVIT_PRESSURE_SP) ]TON(P_800C_CAVIT_VENT_START_DLA_TMR,?,?);
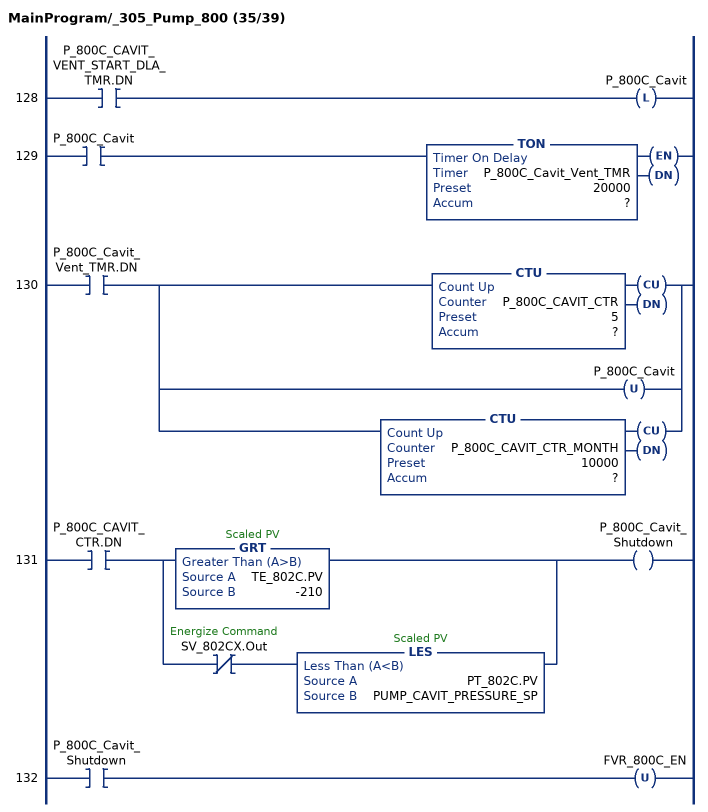
   128: XIC(P_800C_CAVIT_VENT_START_DLA_TMR.DN)OTL(P_800C_Cavit);
   129: XIC(P_800C_Cavit)TON(P_800C_Cavit_Vent_TMR,?,?);
   130: XIC(P_800C_Cavit_Vent_TMR.DN)[CTU(P_800C_CAVIT_CTR,?,?) ,OTU(P_800C_Cavit) ,CTU(P_800C_CAVIT_CTR_MONTH,?,?) ];
   131: XIC(P_800C_CAVIT_CTR.DN)[GRT(TE_802C.PV,-210) ,XIO(SV_802CX.Out) LES(PT_802C.PV,PUMP_CAVIT_PRESSURE_SP) ]OTE(P_800C_Cavit_Shutdown);
   132: XIC(P_800C_Cavit_Shutdown)OTU(FVR_800C_EN);
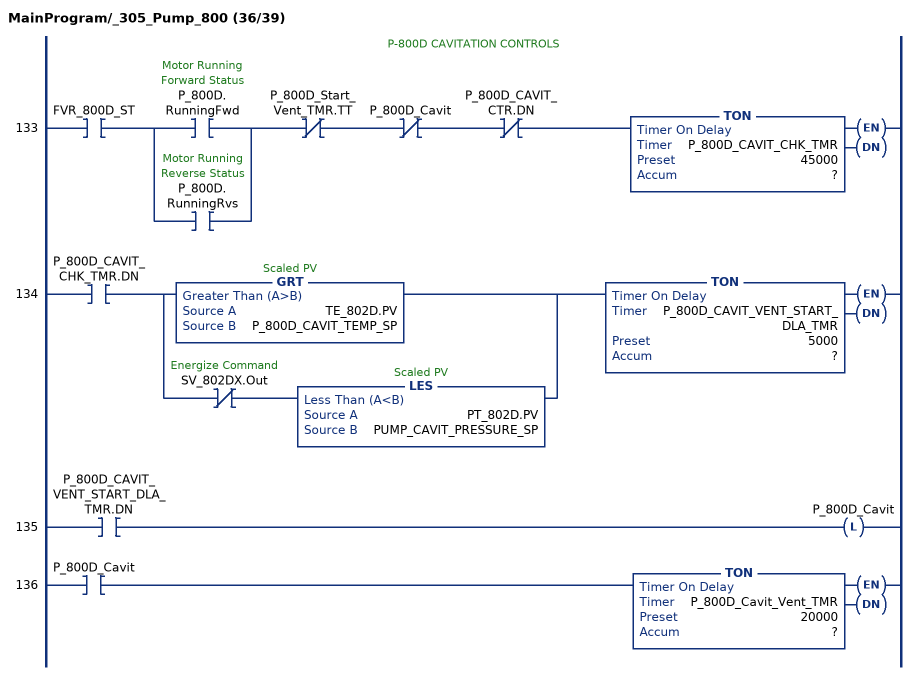
   // P-800D CAVITATION CONTROLS
   133: XIC(FVR_800D_ST)[XIC(P_800D.RunningFwd) ,XIC(P_800D.RunningRvs) ]XIO(P_800D_Start_Vent_TMR.TT)XIO(P_800D_Cavit)XIO(P_800D_CAVIT_CTR.DN)TON(P_800D_CAVIT_CHK_TMR,?,?);
   134: XIC(P_800D_CAVIT_CHK_TMR.DN)[GRT(TE_802D.PV,P_800D_CAVIT_TEMP_SP) ,XIO(SV_802DX.Out) LES(PT_802D.PV,PUMP_CAVIT_PRESSURE_SP) ]TON(P_800D_CAVIT_VENT_START_DLA_TMR,?,?);
   135: XIC(P_800D_CAVIT_VENT_START_DLA_TMR.DN)OTL(P_800D_Cavit);
   136: XIC(P_800D_Cavit)TON(P_800D_Cavit_Vent_TMR,?,?);
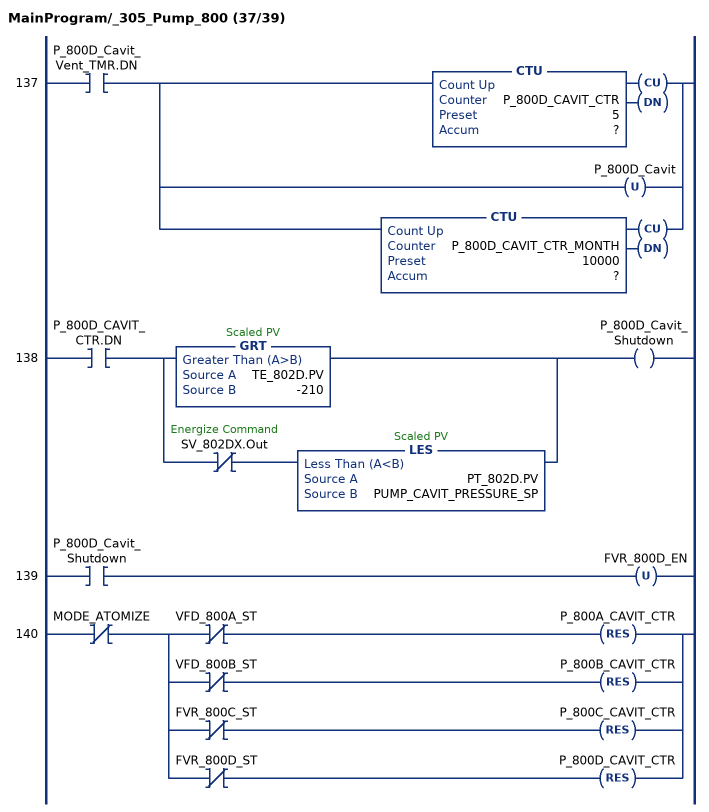
   137: XIC(P_800D_Cavit_Vent_TMR.DN)[CTU(P_800D_CAVIT_CTR,?,?) ,OTU(P_800D_Cavit) ,CTU(P_800D_CAVIT_CTR_MONTH,?,?) ];
   138: XIC(P_800D_CAVIT_CTR.DN)[GRT(TE_802D.PV,-210) ,XIO(SV_802DX.Out) LES(PT_802D.PV,PUMP_CAVIT_PRESSURE_SP) ]OTE(P_800D_Cavit_Shutdown);
   139: XIC(P_800D_Cavit_Shutdown)OTU(FVR_800D_EN);
   140: XIO(MODE_ATOMIZE)[XIO(VFD_800A_ST) RES(P_800A_CAVIT_CTR) ,XIO(VFD_800B_ST) RES(P_800B_CAVIT_CTR) ,XIO(FVR_800C_ST) RES(P_800C_CAVIT_CTR) ,XIO(FVR_800D_ST) RES(P_800D_CAVIT_CTR) ];
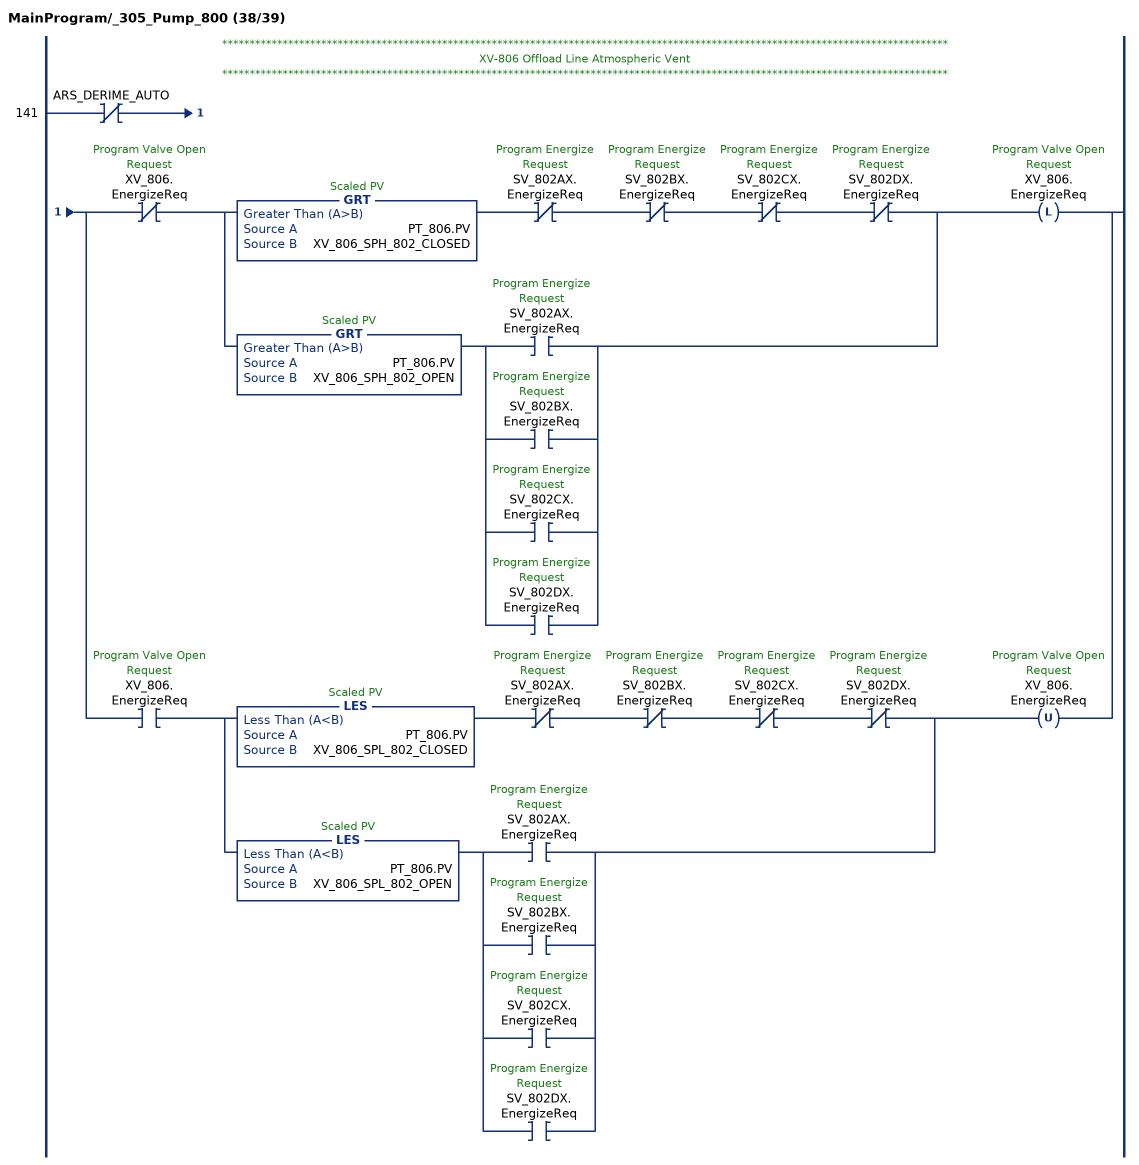
   // ************************************************************************************************************************************
   // XV-806 Offload Line Atmospheric Vent
   // ************************************************************************************************************************************
   141: XIO(ARS_DERIME_AUTO)[XIO(XV_806.EnergizeReq) [GRT(PT_806.PV,XV_806_SPH_802_CLOSED) XIO(SV_802AX.EnergizeReq) XIO(SV_802BX.EnergizeReq) XIO(SV_802CX.EnergizeReq) XIO(SV_802DX.EnergizeReq) ,GRT(PT_806.PV,XV_806_SPH_802_OPEN) [XIC(SV_802AX.EnergizeReq) ,XIC(SV_802BX.EnergizeReq) ,XIC(SV_802CX.EnergizeReq) ,XIC(SV_802DX.EnergizeReq) ] ] OTL(XV_806.EnergizeReq) ,XIC(XV_806.EnergizeReq) [LES(PT_806.PV,XV_806_SPL_802_CLOSED) XIO(SV_802AX.EnergizeReq) XIO(SV_802BX.EnergizeReq) XIO(SV_802CX.EnergizeReq) XIO(SV_802DX.EnergizeReq) ,LES(PT_806.PV,XV_806_SPL_802_OPEN) [XIC(SV_802AX.EnergizeReq) ,XIC(SV_802BX.EnergizeReq) ,XIC(SV_802CX.EnergizeReq) ,XIC(SV_802DX.EnergizeReq) ] ] OTU(XV_806.EnergizeReq) ];
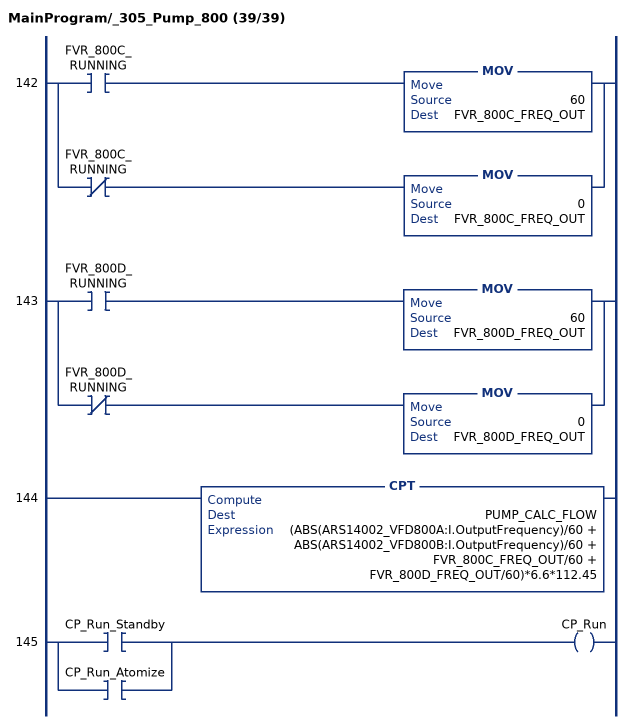
   142: [XIC(FVR_800C_RUNNING) MOV(60,FVR_800C_FREQ_OUT) ,XIO(FVR_800C_RUNNING) MOV(0,FVR_800C_FREQ_OUT) ];
   143: [XIC(FVR_800D_RUNNING) MOV(60,FVR_800D_FREQ_OUT) ,XIO(FVR_800D_RUNNING) MOV(0,FVR_800D_FREQ_OUT) ];
   144: CPT(PUMP_CALC_FLOW,(ABS(ARS14002_VFD800A:I.OutputFrequency)/60 + ABS(ARS14002_VFD800B:I.OutputFrequency)/60 + FVR_800C_FREQ_OUT/60 + FVR_800D_FREQ_OUT/60)*6.6*112.45);
   145: [XIC(CP_Run_Standby) ,XIC(CP_Run_Atomize) ]OTE(CP_Run);
END_ROUTINE
